// TIA Portal V19 export
VAR_GLOBAL   // PLC tag table "HMI conveyor"
   ConveyorOn AT %M10.0 : Bool;
   ConveyorMoving AT %M10.1 : Bool;
   Conveyor_MPM AT %MW12 : Int;
   Conveyor_Max_MPM AT %MW14 : Int;
   Start_System_HMI AT %M20.0 : Bool;
   Stop_System_HMI AT %M20.1 : Bool;
   Reset_System_HMI AT %M20.2 : Bool;
   OS1 AT %M10.2 : Bool;
   ARM_MPM AT %MW34 : Int;
   OS11 AT %M74.3 : Bool;
END_VAR
